// TIA Portal V20 export
TYPE "zd_SCS_ModeBox_InOut"
// stored: Access Published, IsFailsafeCompliant true, Namespace Safety
   STRUCT
      SCSInput : "Safety.zd_SCS_ModeBox_Inputs";
      FaultReset : Bool;
      GuardsOK : Bool;
      AllMotionOFF : Bool;
      SCS1Outputs : "Safety.zd_SCS_ModeBox_Outputs";
      SCSOutputsLT : "Safety.zd_SCS_ModeBox_OutputsLT";
      HazardsRemoved { S7_SetPoint := 'True'} : Bool;
      PendantReqHazControl : Bool;
      MotionsStopped : Bool;
      Faulted : Bool;
      AckReq : Bool;
   END_STRUCT;
END_TYPE
